Fanuc KAREL source: kc00003.KL

-- PROVISIONAL review KL for V1013-1; original PC SHA256 8fbcc92197f8d2484ba9db6e51be7fb9bd11c5ef7490198c9614454630d6ab0f
-- Incomplete behavior may be omitted. Consult companion uncertainty JSON. Do not deploy.
PROGRAM KC00003
%NOLOCKGROUP
BEGIN
  -- UNRESOLVED_PC offsets 5-33; opcodes 27,22,22,22,22,31
  -- UNRESOLVED_PC offsets 38-42; opcodes 7F
END KC00003
